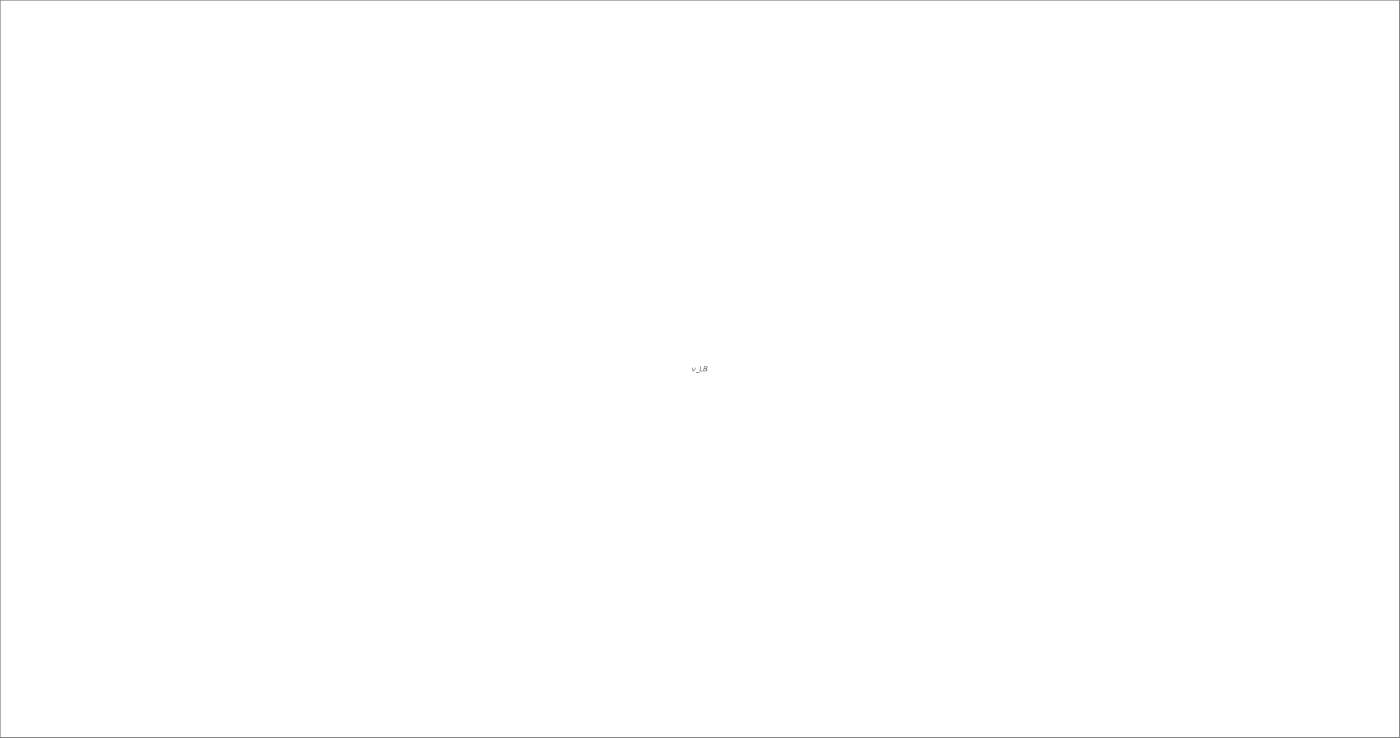
VISUALIZATION visu_LB  // 2048x1080
    TabControl (0,0 2048x1080)
        shows v_LB(dIO_LB := GVL.lb[G_HMI.iLb])
        shows Axis_HMI(st_axis_HMI := st_mcAxis[EN_Axis.Grip_axis])
        shows v_IO_LC(dIO_LC := GVL.lc[G_HMI.iLc])
        shows v_IO_LC()
        shows v_lc(dIO_LC := GVL.lc[1])
        [6]: TabTitle=Gripper
        [1]: AxisHMI=gantrybase.st_mcAxis[EN_Axis.Y], mcAxis=gantrybase.mcAxis[EN_Axis.Y], Error=gantrybase.mcAxis[EN_Axis.Y].xError
        [2]: AxisHMI=gantrybase.st_mcAxis[EN_Axis.Z], mcAxis=gantrybase.mcAxis[EN_Axis.Z], Error=gantrybase.mcAxis[EN_Axis.Z].xError
        p699000190: gantrybase.st_mcAxis[EN_Axis.X]
        p2837713833: gantrybase.mcAxis[EN_Axis.Z].sAxisName
        p520277221: gantrybase.mcAxis[EN_Axis.X].xError
        p3331604638: gantrybase.st_mcAxis[EN_Axis.Z]
        p1813558639: gantrybase.mcAxis[EN_Axis.Z].xError
        p1563495665: gantrybase.st_mcAxis[EN_Axis.Y]
        p2070126892: gantrybase.mcAxis[EN_Axis.Y].xError
        p3435970784: gantrybase.mcAxis[EN_Axis.X]
        p2829954345: gantrybase.mcAxis[EN_Axis.Y]
        p3218520426: gantrybase.mcAxis[EN_Axis.Z]
        p4285860315: GVL.rem[G_HMI.iReM]
        p1681814995: GVL.lc[0]
END_VISUALIZATION

(* stored: Version 1.1.0.1, ProductVersion 3.1.4024.12
   Visu visu_LB: Id {87e7f9fd-188c-400a-b88a-cf1f747a1108} *)
